ORGANIZATION_BLOCK "05_MOD_ERR"
{ S7_Optimized_Access := 'FALSE' }
VERSION : 0.1
   VAR_TEMP
      OB122_EV_CLASS : Byte;
      OB122_SW_FLT : Byte;
      OB122_PRIORITY : Byte;
      OB122_OB_NUMBR : Byte;
      OB122_BLK_TYPE : Byte;
      OB122_MEM_AREA : Byte;
      OB122_MEM_ADDR : Word;
      OB122_BLK_NUM : Word;
      OB122_PRG_ADDR : Word;
      OB122_DATE_TIME : Date_And_Time;
   END_VAR


BEGIN
NETWORK
TITLE =


END_ORGANIZATION_BLOCK

